TYPE Udt_CM_Actuator2State :
STRUCT
	PI_MANUAL :BOOL;
	PI_AUTO : BOOL;
	PI_HMI_HAND : BOOL;
	
	PI_AlarmHigh_Enable : BOOL;
	PI_AlarmLow_Enable : BOOL;
	
	PI_Alarm_Ack_H : BOOL;
	PI_Alarm_Ack_L : BOOL;
	
	PI_Interlock : BOOL;
	PO_Interlocked : BOOL;
	
	PO_ALARM_H : BOOL;
	PO_ALARM_L : BOOL;
	
	PO_HMI_HAND_ON: BOOL;
	PO_AUTO_ON : BOOL;
	PO_MANUAL_ON : BOOL;
	PO_ON : BOOL;
	PO_OFF :BOOL;
	
	
END_STRUCT
END_TYPE

(* stored: Version 1.1.0.1, ProductVersion 3.1.4024.13
   DUT Udt_CM_Actuator2State: Id {e1a01a7e-e03f-4361-bf76-13a6b244c793} *)
